TYPE trafficlight_transitions_typ :
STRUCT
	power_on_Done :BOOL;
	yellow_Done: BOOL;
	green_Done: BOOL;
	red_Done:BOOL;
	blinkON_Done: BOOL;
	blinkOFF_Done: BOOL;
	power_down_ack: BOOL;
	
END_STRUCT
END_TYPE

(* stored: Version 1.1.0.1
   DUT trafficlight_transitions_typ: Id {8b37bf8b-7713-466a-a6d9-a46557be3c8d} *)
